// TIA Portal project "Analytic Process Control2_V16" (V16)

(* hardware
DEVICE "S7-1200 station_2"  S7-1200 Station
   slot 0: "Rack_0"  S7-1200 Rack  Rack  V1.0
   slot 1: "PLC_1"  CPU 1214C DC/DC/DC  6ES7 214-1AG40-0XB0  V4.4
   slot 2: "AI 4x13BIT/AQ 2x14BIT_1"  6ES7 234-4HE32-0XB0  V2.0
DEVICE "HMI_1"  KTP700 Basic PN
   slot 0: "KTP700 Basic PN"  KTP700 Basic PN  6AV2 123-2GB03-0AX0  14.0.1.0
   slot 1: "HMI_RT_1"  KTP700 Basic PN  6AV2 123-2GB03-0AX0  14.0.1.0
   slot 5: "HMI_1.IE_CP_1"  PROFINET Interface  14.0.1.0
      slot 1: "PROFINET Interface_1"  PROFINET Interface
         slot 1: "Port_1"  Port
*)

// ===== PLC "PLC_1"  CPU 1214C DC/DC/DC =====

VAR_GLOBAL   // PLC tag table "Default tag table"
   "SetPoint" AT %MD128 : Real;
   "pH sensor input" AT %IW98 : Int;
   "PID out" AT %MD124 : Real;
   "Scaled pH input" AT %MD120 : Real;
   "Tag_1" AT %MD116 : Real;
   "Tag_2" AT %MD112 : Real;
   "Metering Pump Analog Output" AT %QW96 : Int;
   "Tag_3" AT %IW96 : Int;
   "Tag_4" AT %MD108 : Real;
   "Scaled Pressure reading" AT %MD104 : Real;
   "tank full" AT %M0.0 : Bool;
   "Low level switch" AT %I1.0 : Bool;
   "Circulation pump" AT %Q0.4 : Bool;
   "Start" AT %M0.2 : Bool;
   "Stop" AT %M0.3 : Bool;
   "Sys Run" AT %M0.1 : Bool;
   "High level swich" AT %I0.1 : Bool;
   "Tank outlet Valve" AT %Q0.7 : Bool;
   "tank level" AT %MD96 : Real;
   "tank inlet valve" AT %Q0.6 : Bool;
   "Agitator motor" AT %Q0.5 : Bool;
END_VAR

VAR_GLOBAL   // PLC tag table "NX_Tags"
   "NX_AgitatorMotor" AT %M1.0 : Bool;
   "NX_CirculationPump" AT %M1.1 : Bool;
   "NX_InletValve" AT %M1.2 : Bool;
   "NX_OutletValve" AT %M1.3 : Bool;
END_VAR

DATA_BLOCK "Data_block_1"   // DB3
{ S7_Optimized_Access := 'FALSE' }
VERSION : 0.1
   VAR
      SetPoint : Real;
   END_VAR
BEGIN
END_DATA_BLOCK

FUNCTION "Analog input processing" : Void   // FC1, LAD
{ S7_Optimized_Access := 'TRUE' }
VERSION : 0.1
BEGIN

REGION Network 1
   // pH meter input normalised and scaled to get the real input. this input used as an input in the control PID block
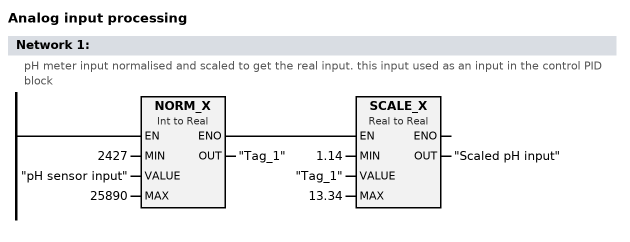
   RUNG wire#powerrail
      { S7_Templates := "[SrcType := Int, DestType := Real]" } Normalize(min := 2427, value := "pH sensor input", max := 25890, out => "Tag_1")
      { S7_Templates := "[SrcType := Real, DestType := Real]" } Scale(min := 1.14, value := "Tag_1", max := 13.34, out => "Scaled pH input")
   END_RUNG
   // the same network as SCL:
   "Tag_1" := NORM_X(MIN := 2427, VALUE := "pH sensor input", MAX := 25890);
   "Scaled pH input" := SCALE_X(MIN := 1.14, VALUE := "Tag_1", MAX := 13.34);
END_REGION
END_FUNCTION

FUNCTION "Analog Output Processsing" : Void   // FC2, LAD
{ S7_Optimized_Access := 'TRUE' }
VERSION : 0.1
BEGIN

REGION Network 1
   // PID compact block output normalised and scaled to machine values.
   // The output fed to the flow control valve analog output channel to the Metering pump. ( doses the Reactor tank with a basic solution when pH is lower than Setpoint)
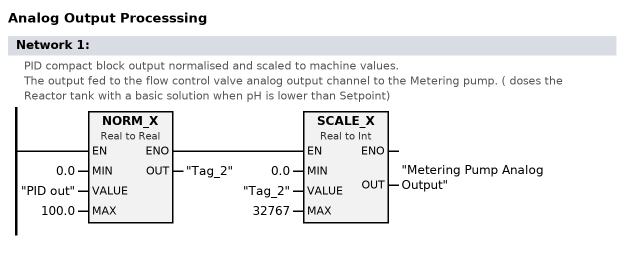
   RUNG wire#powerrail
      { S7_Templates := "[SrcType := Real, DestType := Real]" } Normalize(min := 0.0, value := "PID out", max := 100.0, out => "Tag_2")
      { S7_Templates := "[SrcType := Real, DestType := Int]" } Scale(min := 0.0, value := "Tag_2", max := 32767, out => "Metering Pump Analog Output")
   END_RUNG
   // the same network as SCL:
   "Tag_2" := NORM_X(MIN := 0.0, VALUE := "PID out", MAX := 100.0);
   "Metering Pump Analog Output" := SCALE_X(MIN := 0.0, VALUE := "Tag_2", MAX := 32767);
END_REGION
END_FUNCTION

FUNCTION "Level" : Void   // FC3, LAD
TITLE = Level Control block
{ S7_Optimized_Access := 'TRUE' }
VERSION : 0.1
// Influent and Effluent flows set such that the Reactor tank always remains full.
BEGIN

REGION Network 1: Input processing
   // Normalisation and scaling of the pressure sensor reading.
   // outputs the pressure reading.
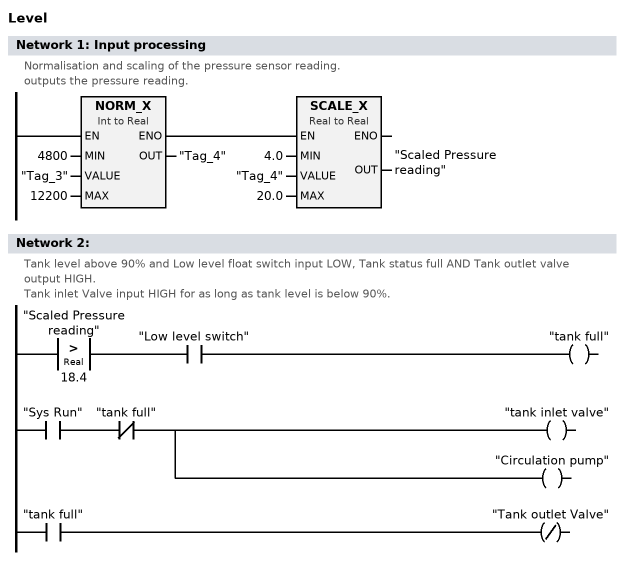
   RUNG wire#powerrail
      { S7_Templates := "[SrcType := Int, DestType := Real]" } Normalize(min := 4800, value := "Tag_3", max := 12200, out => "Tag_4")
      { S7_Templates := "[SrcType := Real, DestType := Real]" } Scale(min := 4.0, value := "Tag_4", max := 20.0, out => "Scaled Pressure reading")
   END_RUNG
   // the same network as SCL:
   "Tag_4" := NORM_X(MIN := 4800, VALUE := "Tag_3", MAX := 12200);
   "Scaled Pressure reading" := SCALE_X(MIN := 4.0, VALUE := "Tag_4", MAX := 20.0);
END_REGION

REGION Network 2
   // Tank level above 90% and Low level float switch input LOW, Tank status full AND Tank outlet valve output HIGH.
   // Tank inlet Valve input HIGH for as long as tank level is below 90%.
   RUNG wire#powerrail
      { S7_Templates := "SrcType := Real" } GT_Contact(in1 := "Scaled Pressure reading", in2 := 18.4)
      Contact( "Low level switch" )
      Coil( "tank full" )
   END_RUNG
   RUNG wire#powerrail
      Contact( "Sys Run" )
      I_Contact( "tank full" )
      wire#w1
      Coil( "tank inlet valve" )
   END_RUNG
   RUNG wire#w1
      Coil( "Circulation pump" )
   END_RUNG
   RUNG wire#powerrail
      Contact( "tank full" )
      I_Coil( "Tank outlet Valve" )
   END_RUNG
   // the same network as SCL:
   "tank full" := ("Scaled Pressure reading" > 18.4) AND "Low level switch";
   "tank inlet valve" := "Sys Run" AND NOT "tank full";
   "Circulation pump" := "tank inlet valve";
   "Tank outlet Valve" := NOT "tank full";
END_REGION
END_FUNCTION

FUNCTION "TIA to NX" : Void   // FC4, LAD
{ S7_Optimized_Access := 'TRUE' }
VERSION : 0.1
BEGIN

REGION Network 1
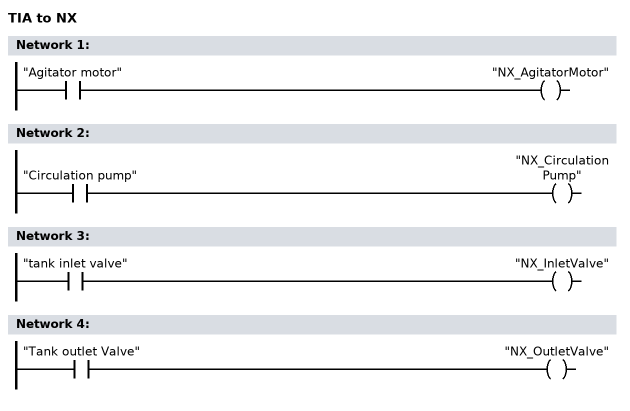
   RUNG wire#powerrail
      Contact( "Agitator motor" )
      Coil( "NX_AgitatorMotor" )
   END_RUNG
   // the same network as SCL:
   "NX_AgitatorMotor" := "Agitator motor";
END_REGION

REGION Network 2
   RUNG wire#powerrail
      Contact( "Circulation pump" )
      Coil( "NX_CirculationPump" )
   END_RUNG
   // the same network as SCL:
   "NX_CirculationPump" := "Circulation pump";
END_REGION

REGION Network 3
   RUNG wire#powerrail
      Contact( "tank inlet valve" )
      Coil( "NX_InletValve" )
   END_RUNG
   // the same network as SCL:
   "NX_InletValve" := "tank inlet valve";
END_REGION

REGION Network 4
   RUNG wire#powerrail
      Contact( "Tank outlet Valve" )
      Coil( "NX_OutletValve" )
   END_RUNG
   // the same network as SCL:
   "NX_OutletValve" := "Tank outlet Valve";
END_REGION
END_FUNCTION

ORGANIZATION_BLOCK "Main"   // OB1, LAD, ProgramCycle
TITLE = "Main Program Sweep (Cycle)"
{ S7_Optimized_Access := 'TRUE' }
VERSION : 0.1
   VAR_INPUT
      Initial_Call : Bool;   // Initial call of this OB
      Remanence : Bool;   // =True, if remanent data are available
   END_VAR
BEGIN

REGION Network 1: Start up conditions
   // Start Input HIGH AND Stop imput HIGH AND low level float switch HIGH, System run conditions ,met.
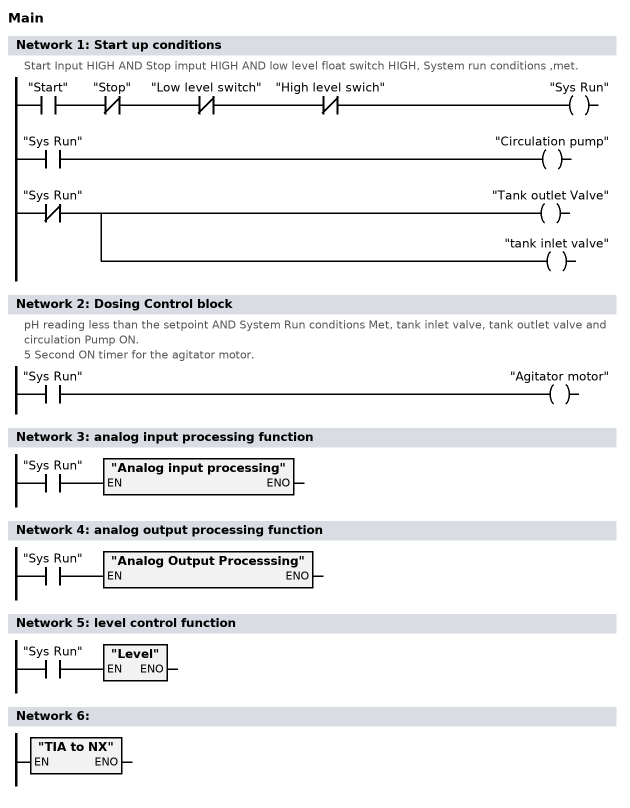
   RUNG wire#powerrail
      Contact( "Start" )
      I_Contact( "Stop" )
      I_Contact( "Low level switch" )
      I_Contact( "High level swich" )
      Coil( "Sys Run" )
   END_RUNG
   RUNG wire#powerrail
      Contact( "Sys Run" )
      Coil( "Circulation pump" )
   END_RUNG
   RUNG wire#powerrail
      I_Contact( "Sys Run" )
      wire#w1
      Coil( "Tank outlet Valve" )
   END_RUNG
   RUNG wire#w1
      Coil( "tank inlet valve" )
   END_RUNG
   // the same network as SCL:
   "Sys Run" := "Start" AND NOT "Stop" AND NOT "Low level switch" AND NOT "High level swich";
   "Circulation pump" := "Sys Run";
   "Tank outlet Valve" := NOT "Sys Run";
   "tank inlet valve" := NOT "Sys Run";
END_REGION

REGION Network 2: Dosing Control block
   // pH reading less than the setpoint AND System Run conditions Met, tank inlet valve, tank outlet valve and circulation Pump ON.
   // 5 Second ON timer for the agitator motor.
   RUNG wire#powerrail
      Contact( "Sys Run" )
      Coil( "Agitator motor" )
   END_RUNG
   // the same network as SCL:
   "Agitator motor" := "Sys Run";
END_REGION

REGION Network 3: analog input processing function
   RUNG wire#powerrail
      Contact( "Sys Run" )
      "Analog input processing"()
   END_RUNG
   // the same network as SCL:
   IF "Sys Run" THEN "Analog input processing"(); END_IF;
END_REGION

REGION Network 4: analog output processing function
   RUNG wire#powerrail
      Contact( "Sys Run" )
      "Analog Output Processsing"()
   END_RUNG
   // the same network as SCL:
   IF "Sys Run" THEN "Analog Output Processsing"(); END_IF;
END_REGION

REGION Network 5: level control function
   RUNG wire#powerrail
      Contact( "Sys Run" )
      "Level"()
   END_RUNG
   // the same network as SCL:
   IF "Sys Run" THEN "Level"(); END_IF;
END_REGION

REGION Network 6
   RUNG wire#powerrail
      "TIA to NX"()
   END_RUNG
   // the same network as SCL:
   "TIA to NX"();
END_REGION
END_ORGANIZATION_BLOCK

ORGANIZATION_BLOCK "Cyclic interrupt(pH)"   // OB30, LAD, CyclicInterrupt
TITLE = PID compact block
{ S7_Optimized_Access := 'TRUE' }
VERSION : 0.1
// Checks the pH reading against the setpoint and provides an output corresponding the the corrective action i.e. opening raiser or reducer agent openings
   VAR_INPUT
      Initial_Call : Bool;   // Initial call of this OB
      Event_Count : Int;   // Events discarded
   END_VAR
BEGIN

REGION Network 1
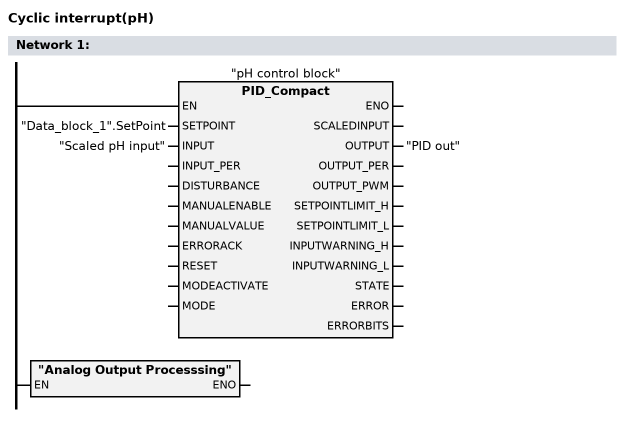
   "pH control block"(Setpoint := "Data_block_1".SetPoint, Input := "Scaled pH input", Output => "PID out");   // PID_Compact
   "Analog Output Processsing"();
END_REGION
END_ORGANIZATION_BLOCK

(* ===== HMI "HMI_RT_1" =====
system functions are stored by id; their names below are inferred from use
connection "HMI_Connection_1": ETHERNET, SMART_S7_1200_OMS

HMI tags "Default tag table"
   "Tag_ScreenNumber" : UInt, internal
   "SetPoint" : Real = PLC SetPoint AT %MD128, 1 s
   "Scaled pH input" : Real = PLC "Scaled pH input" AT %MD120, 1 s
   "Circulation pump" : Bool = PLC "Circulation pump" AT %Q0.4, 1 s
   "Agitator motor" : Bool = PLC "Agitator motor" AT %Q0.5, 1 s
   "tank inlet valve" : Bool = PLC "tank inlet valve" AT %Q0.6, 1 s
   "Tank outlet Valve" : Bool = PLC "Tank outlet Valve" AT %Q0.7, 1 s
   "Start" : Bool = PLC Start AT %M0.2, 1 s
   "Stop" : Bool = PLC Stop AT %M0.3, 1 s

Template "Template_1" 800x480
   Button "Alarms" at 1,52 size 71x50; TextOff 'Alarms'; PictureOff "AlarmDisplay_KTP700_Basic_PN_TR"; PictureOn "AlarmDisplay_KTP700_Basic_PN_TR"
      on Release: function_ef3f5d25("Alarm window_Unacknowledged", -1)
   Button "Template_Button" at 1,106 size 71x50; TextOff 'Text'
   Button "Template_Button_1" at 1,159 size 71x50; TextOff 'Text'
   Button "Template_Button_2" at 1,213 size 71x50; TextOff 'Text'
   Button "Template_Button_3" at 1,267 size 71x50; TextOff 'Text'
   Button "Template_Button_4" at 1,321 size 71x50; TextOff 'Text'
   Button "Template_Button_5" at 1,374 size 71x50; TextOff 'Text'
   Button "Template_Button_6" at 1,428 size 71x50; TextOff 'Text'
   SymbolicIOField "Symbolic_IO_Field_Screen" at 93,9 size 600x33; TextOff '0'; TextOn '1'; TextList "TextList_ScreenNames"
      ProcessValue <- "Tag_ScreenNumber"
      on Change: ActivateScreenByNumber("Tag_ScreenNumber", 0)
   DateTimeField "HmiScreenItemData" at 695,25 size 105x25
   DateTimeField "HmiScreenItemData_1" at 695,0 size 105x25
   GraphicView "Logo" at 0,0 size 91x51; Picture "Logo of HMI_1"

screen "TrendView" 800x480, template "Template_1"
   on GenerateScreen: SetTag("Tag_ScreenNumber", 2)
   TrendView "Trend view_1" at 240,50 size 547x420
   Button "Button_1" at 81,301 size 145x41; TextOff 'SetPoint'
   Button "Button_2" at 80,413 size 142x39; TextOff 'ProcessVariable'
   IOField "I/O field_1" at 81,240 size 143x41; FormatPattern 99
      ProcessValue <- "SetPoint"
   IOField "I/O field_2" at 80,355 size 144x41; FormatPattern 99
      ProcessValue <- "Scaled pH input"
   Switch "Switch_5" at 78,72 size 142x38; TextOn 'ON'; CaptionText 'Switch'; TextOff 'OFF'
      ProcessValue <- "Stop"
   TextField "Text field_13" at 113,116 size 56x27; Text 'STOP'
   Switch "Switch_6" at 79,156 size 142x38; TextOn 'ON'; CaptionText 'Switch'; TextOff 'OFF'
      ProcessValue <- "Start"
   TextField "Text field_14" at 111,202 size 68x27; Text 'START'
*)